TYPE StandardTypesAlias : ST_StandardTypes; END_TYPE

(* stored: Version 1.1.0.1, ProductVersion 3.1.4024.12
   DUT StandardTypesAlias: Id {681ecb69-65b1-4329-a5eb-39829bd27c7f} *)
